// TIA Portal V20 export
// export: Created 2025-12-01T14:56:18.2949384Z, ExportSetting None, DisplayName Totally Integrated Automation Portal, DisplayVersion V20 Update 3, DisplayName TIA Portal Openness, DisplayVersion V20 Update 3, DisplayName TIA Portal Version Control Interface, DisplayVersion V20 Update 3, DisplayName STEP 7 Professional, DisplayVersion V20 Update 3, DisplayName STEP 7 Safety, DisplayVersion V20 Update 2, DisplayName WinCC Basic/Comfort/Advanced, DisplayVersion V20 Update 3, DisplayName WinCC Professional, DisplayVersion V20 Update 3, DisplayName WinCC Unified, DisplayVersion V20 Update 3
TYPE "UDT_VarOmronMX2_V2"
   STRUCT
      Frequecy_Arrival : Bool;
      Control_Status : Bool;
      Reservado_bit_10 : Bool;
      Reservado_bit_11 : Bool;
      Reservado_bit_12 : Bool;
      Reservado_bit_13 : Bool;
      Reservado_bit_14 : Bool;
      Reservado_bit_15 : Bool;
      Reservado_bit_0 : Bool;
      AC_Mains : Bool;
      Ready : Bool;
      Fault : Bool;
      Frecuencia_Ok : Bool;
      Acc_Ok : Bool;
      Dcc_Ok : Bool;
      Alarm : Bool;
      Var_Frecuencia : Int;
      Var_ACC : Int;
      Var_DCC : Int;
      STW_Reserva_Bit8 : Bool;
      STW_Reserva_Bit9 : Bool;
      STW_Reserva_Bit10 : Bool;
      STW_Reserva_Bit11 : Bool;
      STW_Reserva_Bit12 : Bool;
      STW_Reserva_Bit13 : Bool;
      STW_Reserva_Bit14 : Bool;
      STW_Reserva_Bit15 : Bool;
      STW_Var_EnMarcha : Bool;
      STW_Reserva_Bit1 : Bool;
      STW_Reserva_Bit2 : Bool;
      STW_Reserva_Bit3 : Bool;
      STW_Reserva_Bit4 : Bool;
      STW_Reserva_Bit5 : Bool;
      STW_Reserva_Bit6 : Bool;
      STW_Reserva_Bit7 : Bool;
   END_STRUCT;
END_TYPE
